FUNCTION_BLOCK I_WBSD (* Service Interface Function Block Type *)
  (* Standard: ISO 11783-7; Classification: PGN 65096; Function: Wheel-based Speed and Distance WBSD; Description: Copyright (c) 2024 HR Agrartechnik GmbH This program and the accompanying materials are made available under the terms of the Eclipse Public License 2.0 which is available at https://www.eclipse.org/legal/epl-2.0/ SPDX-License-Identifier: EPL-2.0 Message sent by the Tractor ECU on the implement bus on construction and agricultural implements providing to connected systems the current measured wheel-based speed. The message also includes a free-running distance counter, an indication of the direction of travel and the state of the start/stop switch or input. When the ignition key switch is turned off, both the ECU_PWR and PWR have to be maintained to send this message for an additional 2 s. This is not required when the engine is cranking (starting). Accuracies of both wheel-based and ground-based sources can be speed-dependent and degrade at low speeds. Wheel-based information might not be updated at the 100 ms rate at low speeds. https://www.isobus.net/isobus/pGNAndSPN/14648?type=PGN *)
  (* Version 1.0, 2024-07-09, Franz Hoepfinger, HR Agrartechnik GmbH *)
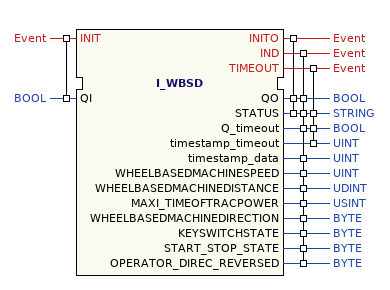
  EVENT_INPUT
    INIT WITH QI; (* Service Initialization *)
  END_EVENT
  EVENT_OUTPUT
    INITO WITH QO, STATUS; (* Initialization Confirm *)
    IND WITH QO, timestamp_data, WHEELBASEDMACHINESPEED, WHEELBASEDMACHINEDISTANCE, MAXI_TIMEOFTRACPOWER, WHEELBASEDMACHINEDIRECTION, KEYSWITCHSTATE, START_STOP_STATE, OPERATOR_DIREC_REVERSED, STATUS, Q_timeout; (* Indication from Resource *)
    TIMEOUT WITH timestamp_timeout, STATUS, Q_timeout;
  END_EVENT
  VAR_INPUT
    QI : BOOL; (* Event Input Qualifier *)
  END_VAR
  VAR_OUTPUT
    QO : BOOL; (* Event Output Qualifier *)
    STATUS : STRING;
    Q_timeout : BOOL;
    timestamp_timeout : UINT;
    timestamp_data : UINT;
    WHEELBASEDMACHINESPEED : UINT; (* Wheel-based machine speed *) {SET_ATTRIBUTE(SPN, 1862)} {SET_ATTRIBUTE(SP_Name, 'Wheel-based machine speed')} {SET_ATTRIBUTE(SP_Position_In_PG, '1-2')} {SET_ATTRIBUTE(SP_Length, 16)} (* 16 bits *) {SET_ATTRIBUTE(Scaling, '0.001 m/s per bit')} {SET_ATTRIBUTE(Offset, )} {SET_ATTRIBUTE(Link, 'https://www.isobus.net/isobus/pGNAndSPN/14642?type=SPN')}
    WHEELBASEDMACHINEDISTANCE : UDINT; (* Wheel-based machine distance *) {SET_ATTRIBUTE(SPN, 1863)} {SET_ATTRIBUTE(SP_Name, 'Wheel-based machine distance')} {SET_ATTRIBUTE(SP_Position_In_PG, '3-6')} {SET_ATTRIBUTE(SP_Length, 16)} (* 32 bits *) {SET_ATTRIBUTE(Scaling, '0.001 m/bit')} {SET_ATTRIBUTE(Offset, )} {SET_ATTRIBUTE(Link, 'https://www.isobus.net/isobus/pGNAndSPN/14643?type=SPN')}
    MAXI_TIMEOFTRACPOWER : USINT; (* Maximum Time of Tractor Power *) {SET_ATTRIBUTE(SPN, 1866)} {SET_ATTRIBUTE(SP_Name, 'Maximum Time of Tractor Power')} {SET_ATTRIBUTE(SP_Position_In_PG, '7')} {SET_ATTRIBUTE(SP_Length, 16)} (* 8 bits *) {SET_ATTRIBUTE(Scaling, '1 min/bit')} {SET_ATTRIBUTE(Offset, )} {SET_ATTRIBUTE(Link, 'https://www.isobus.net/isobus/pGNAndSPN/14644?type=SPN')}
    WHEELBASEDMACHINEDIRECTION : BYTE; (* Wheel-based machine direction *) {SET_ATTRIBUTE(SPN, 1864)} {SET_ATTRIBUTE(SP_Name, 'Wheel-based machine direction')} {SET_ATTRIBUTE(SP_Position_In_PG, '8.1')} {SET_ATTRIBUTE(SP_Length, 16)} (* 2 bits *) {SET_ATTRIBUTE(Scaling, '4 states/2 bit')} {SET_ATTRIBUTE(Offset, )} {SET_ATTRIBUTE(Link, 'https://www.isobus.net/isobus/pGNAndSPN/14645?type=SPN')}
    KEYSWITCHSTATE : BYTE; (* Key switch state *) {SET_ATTRIBUTE(SPN, 1865)} {SET_ATTRIBUTE(SP_Name, 'Key switch state')} {SET_ATTRIBUTE(SP_Position_In_PG, '8.3')} {SET_ATTRIBUTE(SP_Length, 16)} (* 2 bits *) {SET_ATTRIBUTE(Scaling, '4 states/2 bit')} {SET_ATTRIBUTE(Offset, )} {SET_ATTRIBUTE(Link, 'https://www.isobus.net/isobus/pGNAndSPN/14646?type=SPN')}
    START_STOP_STATE : BYTE; (* Implement Start/Stop operations *) {SET_ATTRIBUTE(SPN, 5203)} {SET_ATTRIBUTE(SP_Name, 'Implement Start/Stop operations')} {SET_ATTRIBUTE(SP_Position_In_PG, '8.5')} {SET_ATTRIBUTE(SP_Length, 16)} (* 2 bits *) {SET_ATTRIBUTE(Scaling, '4 states/2 bit')} {SET_ATTRIBUTE(Offset, )} {SET_ATTRIBUTE(Link, 'https://www.isobus.net/isobus/pGNAndSPN/14647?type=SPN')}
    OPERATOR_DIREC_REVERSED : BYTE; (* Operator direction reversed *) {SET_ATTRIBUTE(SPN, 5244)} {SET_ATTRIBUTE(SP_Name, 'Operator direction reversed')} {SET_ATTRIBUTE(SP_Position_In_PG, '8.7')} {SET_ATTRIBUTE(SP_Length, 16)} (* 2 bits *) {SET_ATTRIBUTE(Scaling, '4 states/2 bit')} {SET_ATTRIBUTE(Offset, )} {SET_ATTRIBUTE(Link, 'https://www.isobus.net/isobus/pGNAndSPN/14648?type=SPN')}
  END_VAR
  SERVICE APPLICATION/RESOURCE (* Service Interface Function Block Type *)
    SEQUENCE normal_establishment
      APPLICATION.INIT+(PARAMS) -> RESOURCE.initialize(PARAMS) -> APPLICATION.INITO+();
    END_SEQUENCE
    SEQUENCE unsuccessful_establishment
      APPLICATION.INIT+(PARAMS) -> RESOURCE.initialize(PARAMS) -> APPLICATION.INITO-(STATUS);
    END_SEQUENCE
    SEQUENCE request_confirm
      APPLICATION.REQ+(SD) -> RESOURCE.request(SD) -> APPLICATION.CNF+(RD);
    END_SEQUENCE
    SEQUENCE request_inhibited
      APPLICATION.REQ-(SD) -> APPLICATION.CNF-(STATUS);
    END_SEQUENCE
    SEQUENCE request_error
      APPLICATION.REQ+(SD) -> RESOURCE.request(SD) -> APPLICATION.CNF-(STATUS);
    END_SEQUENCE
    SEQUENCE indication_response
      RESOURCE.indicate(RD) -> APPLICATION.IND+(RD);
      APPLICATION.RSP(QI,SD) -> RESOURCE.response(QI,SD);
    END_SEQUENCE
    SEQUENCE indication_inhibited
      RESOURCE.indicate(RD,QI=FALSE) -> RESOURCE.inhibited();
    END_SEQUENCE
    SEQUENCE error_indication
      RESOURCE.error(STATUS) -> APPLICATION.IND-(STATUS);
    END_SEQUENCE
    SEQUENCE application_initiated_termination
      APPLICATION.INIT-() -> RESOURCE.terminate() -> APPLICATION.INITO-(STATUS);
    END_SEQUENCE
    SEQUENCE resource_initiated_termination
      -> APPLICATION.INITO-(STATUS);
    END_SEQUENCE
  END_SERVICE
END_FUNCTION_BLOCK
